FUNCTION "FC_Action_Ap_Cir_Sous_Broy" : Bool
{ S7_Optimized_Access := 'TRUE' }
VERSION : 0.1
   VAR_IN_OUT
      Broyeur : "S_Broyage";
   END_VAR


BEGIN
	#FC_Action_Ap_Cir_Sous_Broy := TRUE;
END_FUNCTION

